(* Logix 5000 project; controller PruebaIgnition vendor 1 type 14 code 156 rev 30.11; software revision 30.00 *)

TASK MainTask (continuous, watchdog 500 ms) : MainProgram

MODULES
   Local : vendor 1 type 14 code 156 (Compact 0, rev 30.11)
      DIs : 1769-IQ16 (Compact 4, rev 1.1, Input RPI 20 ms)
      DOs : vendor 1 type 7 code 86 (Compact 5, rev 2.1, Output RPI 20 ms)
      AOs : vendor 1 type 10 code 48 (Compact 3, rev 1.1, Output RPI 80 ms)
END_MODULES

VAR_GLOBAL   (* controller tags *)
   BandaG : BOOL;
   BandaP : BOOL;
   C_Box : TIMER := (PRE := 1500);
   Cajas_Grande : INT := 4;
   Cajas_Mediana : INT := 1;
   Cajas_Pequena : INT := 5;
   Ciclo_inicialG : BOOL;
   Ciclo_inicialM : BOOL;
   Ciclo_inicialP : BOOL;
   CounterG : COUNTER := (PRE := 100);
   CounterG2 : COUNTER := (PRE := 100);
   CounterM : COUNTER := (PRE := 100);
   CounterM2 : COUNTER := (PRE := 100);
   CounterP : COUNTER := (PRE := 100);
   CounterP2 : COUNTER := (PRE := 100);
   Etapa_0 : BOOL;
   Etapa_0G : BOOL;
   Etapa_0M : BOOL := 1;
   Etapa_0P : BOOL := 1;
   Etapa_1 : BOOL;
   Etapa_1G : BOOL := 1;
   Etapa_1M : BOOL;
   Etapa_1P : BOOL;
   Etapa_2 : BOOL;
   Etapa_2G : BOOL;
   Etapa_2M : BOOL := 1;
   Etapa_2P : BOOL := 1;
   Etapa_3 : BOOL;
   Etapa_3G : BOOL := 1;
   Etapa_3M : BOOL;
   Etapa_3P : BOOL;
   Etapa_4 : BOOL;
   Etapa_5 : BOOL;
   Etapa_6 : BOOL;
   FaltanG : BOOL;
   FaltanM : BOOL := 1;
   FaltanP : BOOL;
   FaltantesG : INT;
   FaltantesM : DINT;
   FaltantesP : DINT;
   Grande : BOOL;
   Mediano : BOOL;
   PedidoG : BOOL := 1;
   PedidoM : BOOL := 1;
   PedidoP : BOOL := 1;
   Pequeno : BOOL;
   Ph_MotorBandas : ALIAS FOR Local:3:O.Ch0Data;
   PickG : BOOL := 1;
   PickM : BOOL;
   PickP : BOOL;
   Potenciometro : INT := 1000;
   Primer_Ciclo : BOOL;
   Reset : BOOL := 1;
   Send : BOOL;
   SorterLeft : BOOL;
   SorterRight : BOOL;
   Start_btn : BOOL;
   Stop_btn : BOOL;
   Timer_Caja : TIMER := (PRE := 1500);
   TimerG : TIMER := (PRE := 10000);
   TimerM : TIMER := (PRE := 10000);
   TimerP : TIMER := (PRE := 10000);
   V_A_0 : BOOL;
   V_A_1 : BOOL;
   V_A_10 : BOOL;
   V_A_11 : BOOL;
   V_A_13 : BOOL;
   V_A_14 : BOOL := 1;
   V_A_15 : BOOL := 1;
   V_A_2 : BOOL;
   V_A_3 : BOOL;
   V_A_4 : BOOL := 1;
   V_A_5 : BOOL := 1;
   V_A_6 : BOOL := 1;
   V_A_7 : BOOL;
   V_A_8 : BOOL;
   V_A_9 : BOOL;
   V_A_Emit : BOOL;
   V_A_PUSH_G : BOOL;
   V_A_PUSH_M : BOOL := 1;
   V_A_PUSH_P : BOOL := 1;
   V_A_StackG : BOOL := 1;
   V_A_StackM : BOOL;
   V_A_StackP : BOOL;
   V_S_0 : BOOL;
   V_S_1 : BOOL;
   V_S_10 : BOOL;
   V_S_11 : BOOL;
   V_S_12 : BOOL;
   V_S_13 : BOOL;
   V_S_14 : BOOL;
   V_S_16 : BOOL;
   V_S_2 : BOOL;
   V_S_3 : BOOL;
   V_S_4 : BOOL;
   V_S_5 : BOOL;
   V_S_6 : BOOL;
   V_S_7 : BOOL;
   V_S_8 : BOOL;
   V_S_9 : BOOL;
END_VAR

PROGRAM MainProgram   (* main routine MainRoutine *)

ROUTINE Grafcet   (* ladder *)
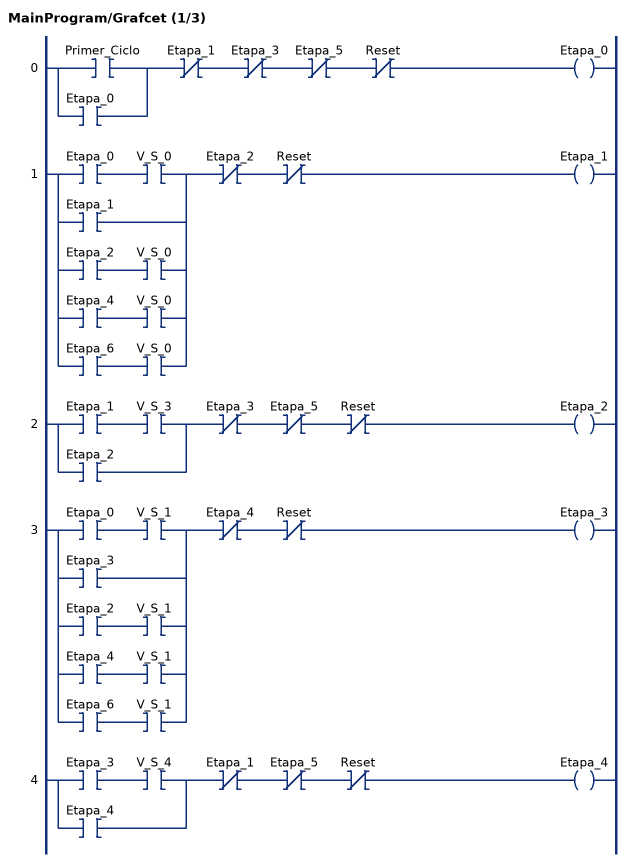
   0: [XIC(Primer_Ciclo) ,XIC(Etapa_0) ]XIO(Etapa_1)XIO(Etapa_3)XIO(Etapa_5)XIO(Reset)OTE(Etapa_0);
   1: [[[[XIC(Etapa_0) XIC(V_S_0) ,XIC(Etapa_1) ] ,XIC(Etapa_2) XIC(V_S_0) ] ,XIC(Etapa_4) XIC(V_S_0) ] ,XIC(Etapa_6) XIC(V_S_0) ]XIO(Etapa_2)XIO(Reset)OTE(Etapa_1);
   2: [XIC(Etapa_1) XIC(V_S_3) ,XIC(Etapa_2) ]XIO(Etapa_3)XIO(Etapa_5)XIO(Reset)OTE(Etapa_2);
   3: [XIC(Etapa_0) XIC(V_S_1) ,XIC(Etapa_3) ,XIC(Etapa_2) XIC(V_S_1) ,XIC(Etapa_4) XIC(V_S_1) ,XIC(Etapa_6) XIC(V_S_1) ]XIO(Etapa_4)XIO(Reset)OTE(Etapa_3);
   4: [XIC(Etapa_3) XIC(V_S_4) ,XIC(Etapa_4) ]XIO(Etapa_1)XIO(Etapa_5)XIO(Reset)OTE(Etapa_4);
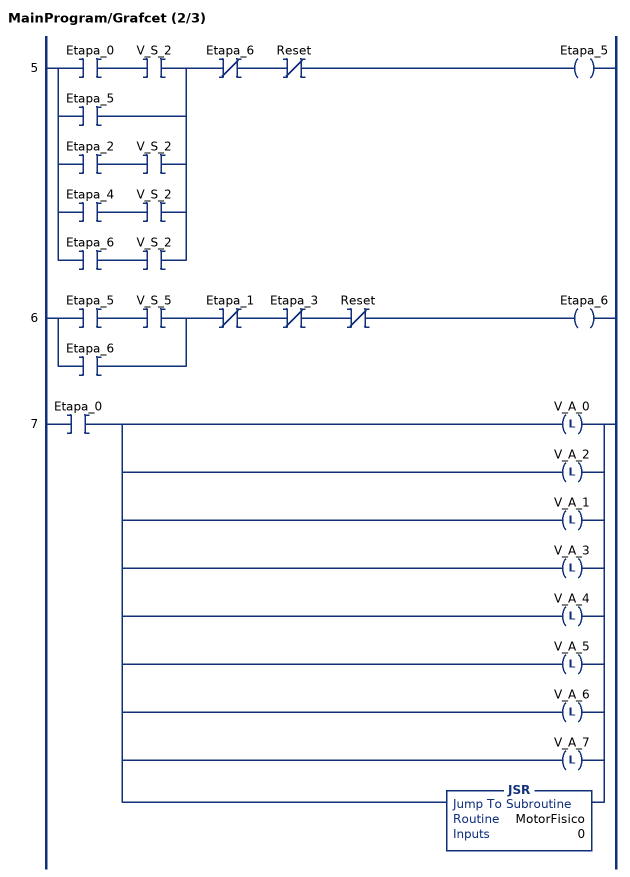
   5: [XIC(Etapa_0) XIC(V_S_2) ,XIC(Etapa_5) ,XIC(Etapa_2) XIC(V_S_2) ,XIC(Etapa_4) XIC(V_S_2) ,XIC(Etapa_6) XIC(V_S_2) ]XIO(Etapa_6)XIO(Reset)OTE(Etapa_5);
   6: [XIC(Etapa_5) XIC(V_S_5) ,XIC(Etapa_6) ]XIO(Etapa_1)XIO(Etapa_3)XIO(Reset)OTE(Etapa_6);
   7: XIC(Etapa_0)[OTL(V_A_0) ,OTL(V_A_2) ,OTL(V_A_1) ,OTL(V_A_3) ,OTL(V_A_4) ,OTL(V_A_5) ,OTL(V_A_6) ,OTL(V_A_7) ,JSR(MotorFisico,0) ];
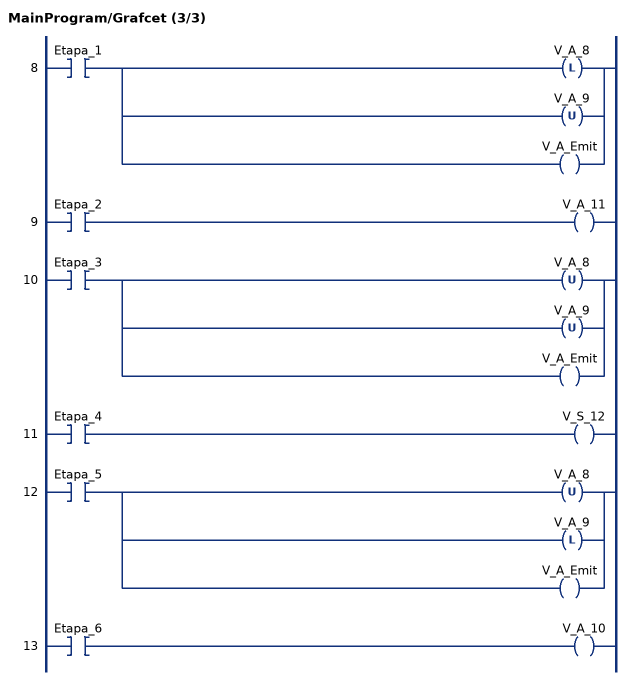
   8: XIC(Etapa_1)[OTL(V_A_8) ,OTU(V_A_9) ,OTE(V_A_Emit) ];
   9: XIC(Etapa_2)OTE(V_A_11);
   10: XIC(Etapa_3)[OTU(V_A_8) ,OTU(V_A_9) ,OTE(V_A_Emit) ];
   11: XIC(Etapa_4)OTE(V_S_12);
   12: XIC(Etapa_5)[OTU(V_A_8) ,OTL(V_A_9) ,OTE(V_A_Emit) ];
   13: XIC(Etapa_6)OTE(V_A_10);
END_ROUTINE

ROUTINE MainRoutine   (* ladder *)
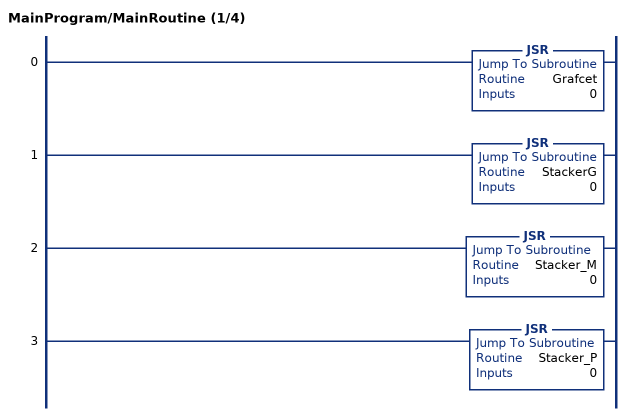
   0: JSR(Grafcet,0);
   1: JSR(StackerG,0);
   2: JSR(Stacker_M,0);
   3: JSR(Stacker_P,0);
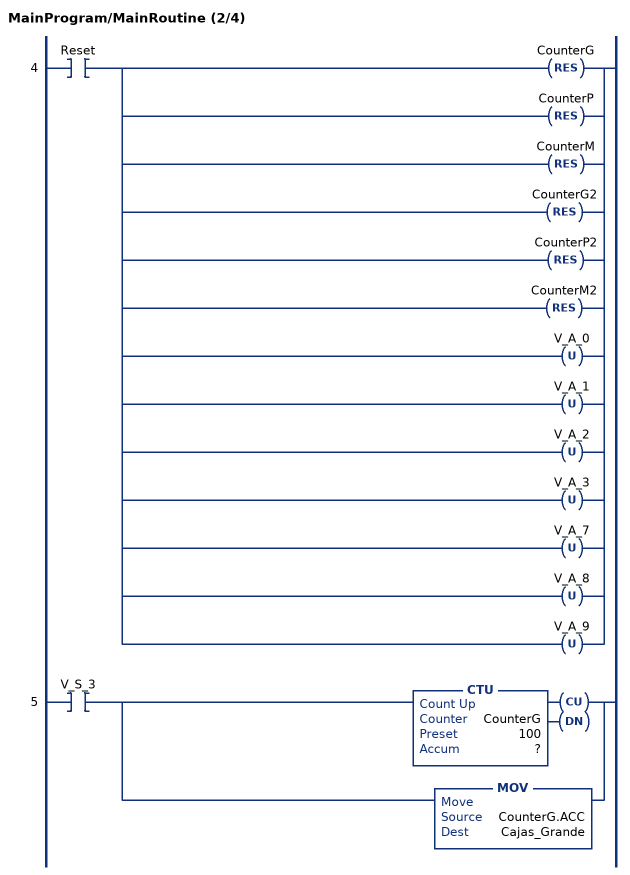
   4: XIC(Reset)[RES(CounterG) ,RES(CounterP) ,RES(CounterM) ,RES(CounterG2) ,RES(CounterP2) ,RES(CounterM2) ,OTU(V_A_0) ,OTU(V_A_1) ,OTU(V_A_2) ,OTU(V_A_3) ,OTU(V_A_7) ,OTU(V_A_8) ,OTU(V_A_9) ];
   5: XIC(V_S_3)[CTU(CounterG,?,?) ,MOV(CounterG.ACC,Cajas_Grande) ];
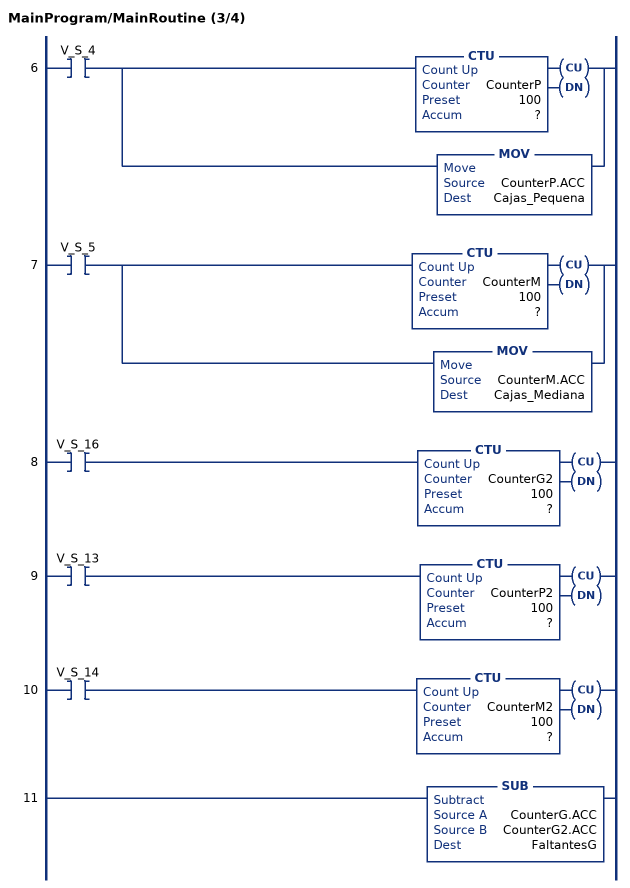
   6: XIC(V_S_4)[CTU(CounterP,?,?) ,MOV(CounterP.ACC,Cajas_Pequena) ];
   7: XIC(V_S_5)[CTU(CounterM,?,?) ,MOV(CounterM.ACC,Cajas_Mediana) ];
   8: XIC(V_S_16)CTU(CounterG2,?,?);
   9: XIC(V_S_13)CTU(CounterP2,?,?);
   10: XIC(V_S_14)CTU(CounterM2,?,?);
   11: SUB(CounterG.ACC,CounterG2.ACC,FaltantesG);
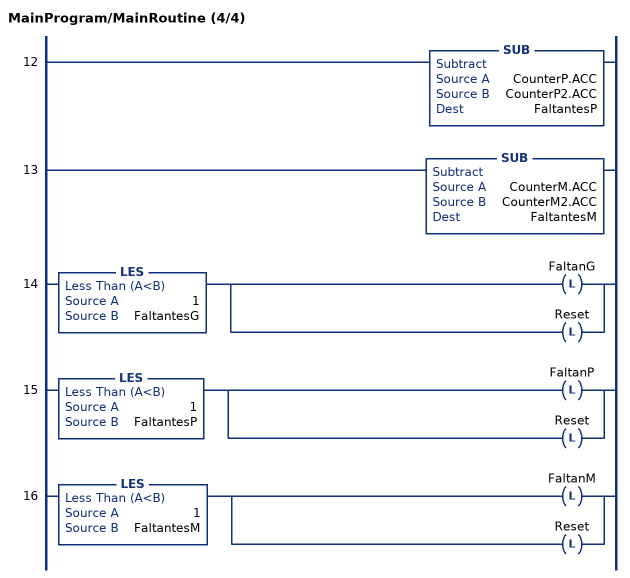
   12: SUB(CounterP.ACC,CounterP2.ACC,FaltantesP);
   13: SUB(CounterM.ACC,CounterM2.ACC,FaltantesM);
   14: LES(1,FaltantesG)[OTL(FaltanG) ,OTL(Reset) ];
   15: LES(1,FaltantesP)[OTL(FaltanP) ,OTL(Reset) ];
   16: LES(1,FaltantesM)[OTL(FaltanM) ,OTL(Reset) ];
END_ROUTINE

ROUTINE MotorFisico   (* ladder *)
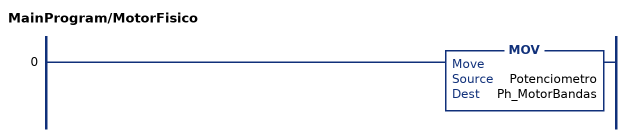
   0: MOV(Potenciometro,Ph_MotorBandas);
END_ROUTINE

ROUTINE Stacker_M   (* ladder *)
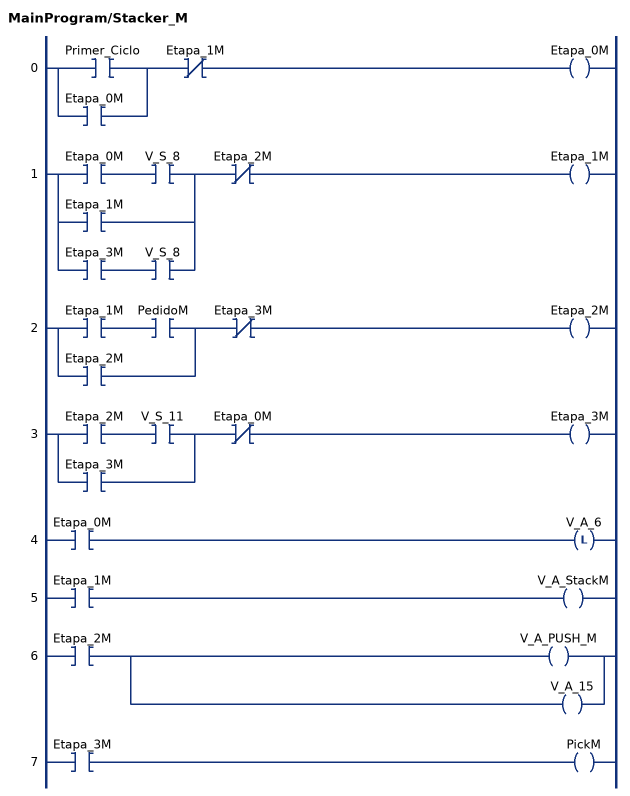
   0: [XIC(Primer_Ciclo) ,XIC(Etapa_0M) ]XIO(Etapa_1M)OTE(Etapa_0M);
   1: [XIC(Etapa_0M) XIC(V_S_8) ,XIC(Etapa_1M) ,XIC(Etapa_3M) XIC(V_S_8) ]XIO(Etapa_2M)OTE(Etapa_1M);
   2: [XIC(Etapa_1M) XIC(PedidoM) ,XIC(Etapa_2M) ]XIO(Etapa_3M)OTE(Etapa_2M);
   3: [XIC(Etapa_2M) XIC(V_S_11) ,XIC(Etapa_3M) ]XIO(Etapa_0M)OTE(Etapa_3M);
   4: XIC(Etapa_0M)OTL(V_A_6);
   5: XIC(Etapa_1M)OTE(V_A_StackM);
   6: XIC(Etapa_2M)[OTE(V_A_PUSH_M) ,OTE(V_A_15) ];
   7: XIC(Etapa_3M)OTE(PickM);
END_ROUTINE

ROUTINE Stacker_P   (* ladder *)
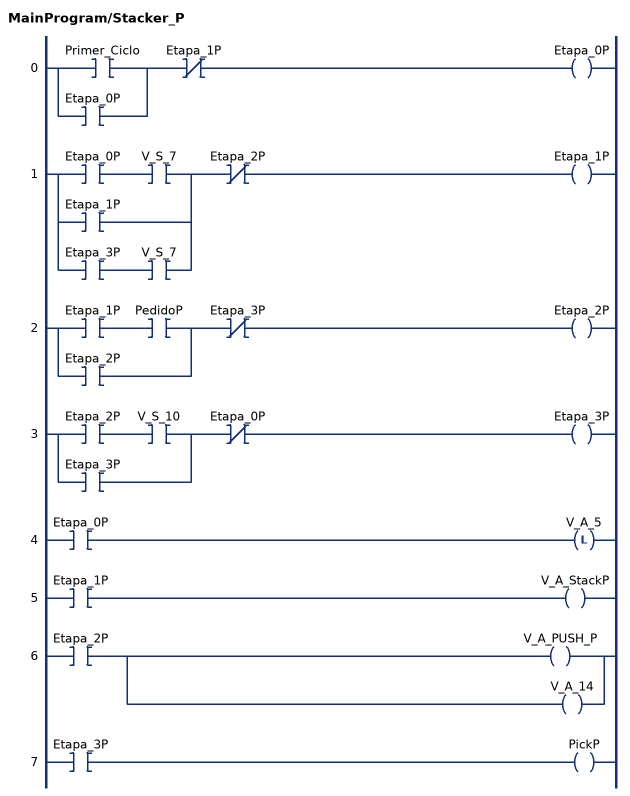
   0: [XIC(Primer_Ciclo) ,XIC(Etapa_0P) ]XIO(Etapa_1P)OTE(Etapa_0P);
   1: [XIC(Etapa_0P) XIC(V_S_7) ,XIC(Etapa_1P) ,XIC(Etapa_3P) XIC(V_S_7) ]XIO(Etapa_2P)OTE(Etapa_1P);
   2: [XIC(Etapa_1P) XIC(PedidoP) ,XIC(Etapa_2P) ]XIO(Etapa_3P)OTE(Etapa_2P);
   3: [XIC(Etapa_2P) XIC(V_S_10) ,XIC(Etapa_3P) ]XIO(Etapa_0P)OTE(Etapa_3P);
   4: XIC(Etapa_0P)OTL(V_A_5);
   5: XIC(Etapa_1P)OTE(V_A_StackP);
   6: XIC(Etapa_2P)[OTE(V_A_PUSH_P) ,OTE(V_A_14) ];
   7: XIC(Etapa_3P)OTE(PickP);
END_ROUTINE

ROUTINE StackerG   (* ladder *)
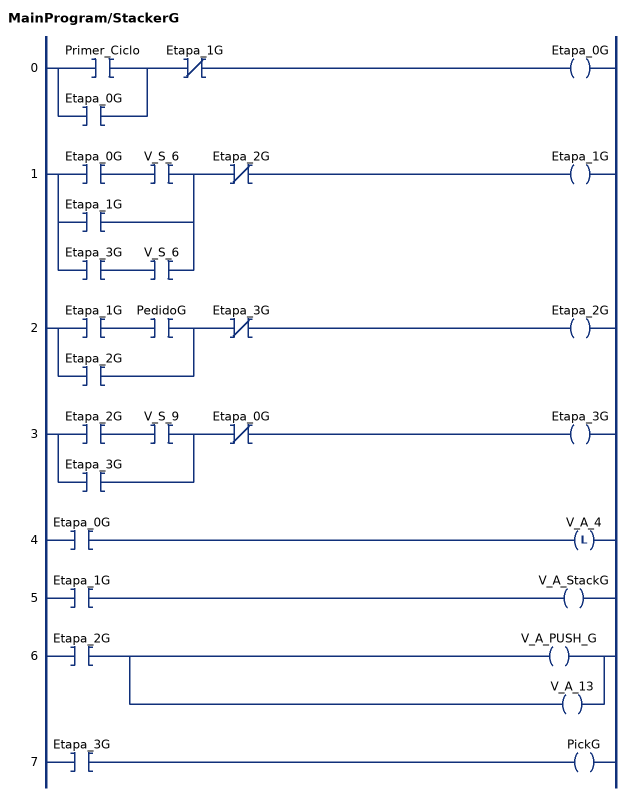
   0: [XIC(Primer_Ciclo) ,XIC(Etapa_0G) ]XIO(Etapa_1G)OTE(Etapa_0G);
   1: [XIC(Etapa_0G) XIC(V_S_6) ,XIC(Etapa_1G) ,XIC(Etapa_3G) XIC(V_S_6) ]XIO(Etapa_2G)OTE(Etapa_1G);
   2: [XIC(Etapa_1G) XIC(PedidoG) ,XIC(Etapa_2G) ]XIO(Etapa_3G)OTE(Etapa_2G);
   3: [XIC(Etapa_2G) XIC(V_S_9) ,XIC(Etapa_3G) ]XIO(Etapa_0G)OTE(Etapa_3G);
   4: XIC(Etapa_0G)OTL(V_A_4);
   5: XIC(Etapa_1G)OTE(V_A_StackG);
   6: XIC(Etapa_2G)[OTE(V_A_PUSH_G) ,OTE(V_A_13) ];
   7: XIC(Etapa_3G)OTE(PickG);
END_ROUTINE
END_PROGRAM
